// TIA Portal V20 export
DATA_BLOCK "DB_AsiSetpoint"   // DB28
// stored: Access Published, MemoryReserve 100, Namespace PackedLine
   VAR
      Line : Struct
         PackedLine : Struct
            DirChange : Struct
               Conveyor : Array[_.minPackedLine.._.maxPackedLine] of Bool;
            END_STRUCT;
            Speed : Struct
               Conveyor : Array[_.minPackedLine.._.maxPackedLine] of Bool;
            END_STRUCT;
         END_STRUCT;
      END_STRUCT;
   END_VAR
BEGIN
END_DATA_BLOCK
